Staubli VAL3: setPoint.pgx

public program setPoint(string x_sPoint)
begin
  //
  sPointName=x_sPoint
end
